ABB RobotStudio station: Paletizado.rspag

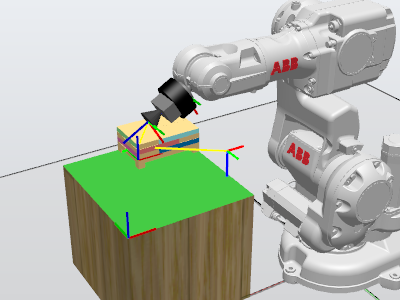
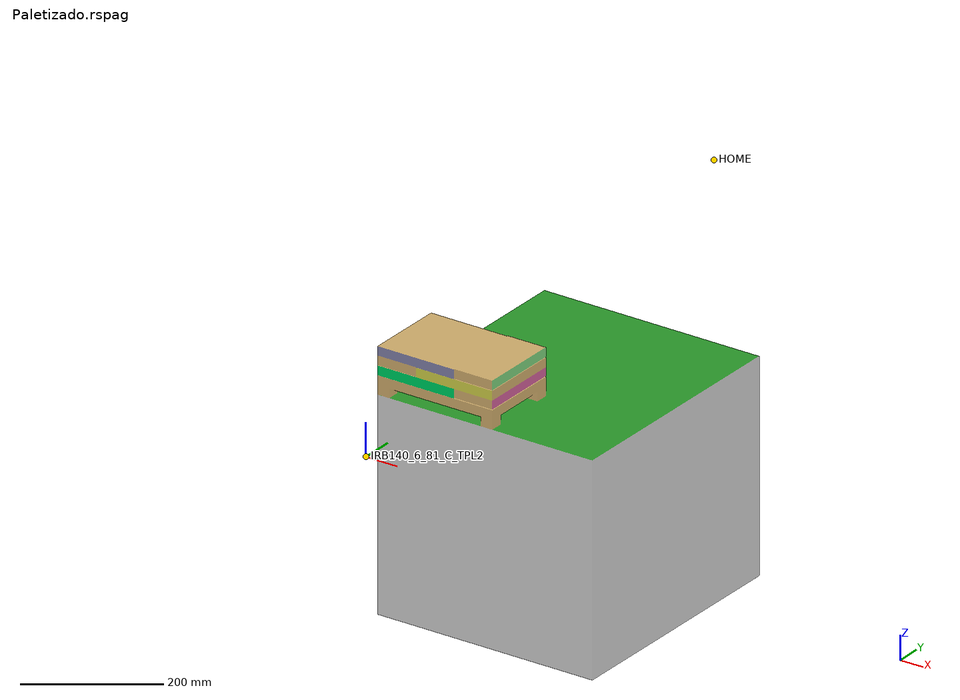
[picture v1: parts stored in the station drawn from their meshes, with robot base, taught points and paths (robot models come from the ABB library and are not in the file)]
--- station ---
Station Paletizado (saved by RobotStudio 25.1.11167.1)
Controller IRB140_6_81_TPL2
  mechanical unit ROB_1: IRB140_6_81_C_TPL2, 6 joints, base frame (0, 0, 0) mm
Layout (positions relative to the parent item):
  - Mesa [part], size 365 x 405 x 340 mm
  - Pallet [part], size 195 x 130 x 30 mm
  - Pieza1 [part] at (0, -275, 60) mm, size 130 x 65 x 15 mm
  - Pieza2 [part] at (729.91, -395, 45.09) mm, rotated rx 0 ry 0 rz 180 deg, size 130 x 65 x 15 mm
  - Pieza3 [part] at (490, 30, 30.97) mm, rotated rx 0 ry 0 rz -90 deg, size 130 x 65 x 15 mm
  - Pieza4 [part] at (795, -395, 0) mm, rotated rx 0 ry 0 rz -180 deg, size 130 x 65 x 15 mm
  - Pieza5 [part] at (65, -275, -15) mm, size 130 x 65 x 15 mm
  - Pieza6 [part] at (305, -700, -29.39) mm, rotated rx 0 ry 0 rz 90 deg, size 130 x 65 x 15 mm
  - Pieza7 [part] at (0, -275, -60) mm, size 130 x 65 x 15 mm
  - Pieza8 [part] at (729.88, -395, -74.88) mm, rotated rx 0 ry 0 rz 180 deg, size 130 x 65 x 15 mm
  - Pieza9 [part] at (490, 30, -88.74) mm, rotated rx 0 ry 0 rz -90 deg, size 130 x 65 x 15 mm
  - Sopapa [mechanism] at (506.29, 0, 679.5) mm, rotated rx 180 ry 60 rz 180 deg
      TCP Sopapa at (0, -5, 103) mm
      links: Sopapa
  - IRB140_6_81_C_TPL2 [mechanism, from %ABB.RobotStudio.Models.IRB140%\IRB140_6_81_C_G_03.rslib] at (0, 0, 0) mm; joint values [0, 0, 0, 0, 0.5236, 0] (rad or m)
Attachment: Sopapa is attached to IRB140_6_81_C_TPL2 / Link6
EventTableEntry 1212: Group=, Trigger=DO_Pinza 1213, Actions=[EventTableActionAttach 1214], Comment=, ActivationMode=2, Cyclic=false
EventTableTriggerIO 1213: IOValue=[1], IRC5Controller=? -1, Operator=0, SignalSource=? -1
EventTableActionAttach 1214: AttachmentParent=Sopapa 1252, AttachmentChild=? -1, MountObject=false, Offset=[X=1, Y=0, Z=0, W=0, X=0, Y=1, Z=0, W=0, X=0, Y=0, Z=1, W=0, X=0, Y=0, Z=0, W=1], FlangeIndext=0, FindNearest=true
EventTableEntry 1219: Group=, Trigger=DO_Pinza 1220, Actions=[EventTableActionDetach 1221], Comment=, ActivationMode=2, Cyclic=false
EventTableTriggerIO 1220: IOValue=[0], IRC5Controller=? -1, Operator=0, SignalSource=? -1
EventTableActionDetach 1221: AttachmentParent=Sopapa 1252, AttachmentChild=? -1
EventTableEntry 2390: Group=, Trigger=DO_SOPAPA 2391, Actions=[EventTableActionAttach 2392], Comment=, ActivationMode=2, Cyclic=false
EventTableTriggerIO 2391: IOValue=[1], IRC5Controller=? -1, Operator=0, SignalSource=IRB140_6_81_TPL2 1258
EventTableActionAttach 2392: AttachmentParent=Sopapa 1252, AttachmentChild=? -1, MountObject=false, Offset=[X=1, Y=0, Z=0, W=0, X=0, Y=1, Z=0, W=0, X=0, Y=0, Z=1, W=0, X=0, Y=0, Z=0, W=1], FlangeIndext=0, FindNearest=true
EventTableEntry 3475: Group=, Trigger=DO_SOPAPA 3476, Actions=[EventTableActionDetach 3477], Comment=, ActivationMode=2, Cyclic=false
EventTableTriggerIO 3476: IOValue=[0], IRC5Controller=? -1, Operator=0, SignalSource=IRB140_6_81_TPL2 1258
EventTableActionDetach 3477: AttachmentParent=Sopapa 1252, AttachmentChild=? -1
Targets, tools, work objects and paths stored in the station and not in the controller backup, written as RAPID:
! task T_ROB1
MODULE Module1
  CONST robtarget PPLACE1_2:=[[32.5,65,0],[0,0.707106781,0.707106781,0],[-1,0,-2,0],[9E+09,9E+09,9E+09,9E+09,9E+09,9E+09]];
  PROC Path_20()
    MoveL PPICK,v1000,z100,Sopapa\WObj:=RMESA;
    MoveL PPICK,v1000,z100,Sopapa\WObj:=RMESA;
    MoveL PPLACE1,v1000,z100,Sopapa\WObj:=RPALET;
    MoveL HOME,v1000,z100,Sopapa\WObj:=wobj0;
    MoveL PPLACE1_2,v1000,z100,Sopapa\WObj:=RPALET;
  ENDPROC
ENDMODULE


--- Backups/IRB140_6_81_TPL2/RAPID/TASK1/PROGMOD/CalibData.mod ---
MODULE CalibData
    TASK PERS wobjdata RPALET:=[FALSE,TRUE,"",[[495,-270,370],[0,0,0,1]],[[0,0,0],[1,0,0,0]]];
    TASK PERS wobjdata RMESA:=[FALSE,TRUE,"",[[665,5,340],[0,0,0,1]],[[0,0,0],[1,0,0,0]]];
ENDMODULE

--- Backups/IRB140_6_81_TPL2/RAPID/TASK1/PROGMOD/Module1.mod ---
MODULE Module1
    !!!!! USAR MAYUSCULAS PARA LAS CONSTANTES
    PERS tooldata Sopapa:=[TRUE,[[0,-5,103],[1,0,0,0]],[0.5,[0,0,40],[1,0,0,0],0,0,0]];
    PERS tooldata Sopapa_caja:=[TRUE,[[0,-5,118],[1,0,0,0]],[0.5,[0,0,40],[1,0,0,0],0,0,0]];
    CONST robtarget PPICK:=[[300,32.5,135],[0,1,0,0],[0,0,0,0],[9E+09,9E+09,9E+09,9E+09,9E+09,9E+09]];
    CONST robtarget PPLACE1:=[[32.5,65,0],[0,-0.707106781,0.707106781,0],[0,0,0,0],[9E+09,9E+09,9E+09,9E+09,9E+09,9E+09]];
    CONST robtarget HOME:=[[595.492267836,-5,628],[0.5,0,0.866025404,0],[0,-1,0,0],[9E+09,9E+09,9E+09,9E+09,9E+09,9E+09]];
    CONST num cant_cajas:=9;
    CONST num h_caja:=15;
    CONST num dx_PPLACE1:=130;
    VAR num CajasEnPalet:=0;

    !***********************************************************
    !
    ! Module:  Module1
    !
    ! Description:
    !   <Insert description here>
    !
    ! Author: CARLOS ISAAC
    !
    ! Version: 1.0
    !
    !***********************************************************


    !***********************************************************
    !
    ! Procedure main
    !
    !   This is the entry point of your program
    !
    !***********************************************************
    PROC main()
        !Add your code here
        VAR num pila:=0; !indica la pila actual de paletizado iniciando en 0
        VAR num caja_pilai:=0; !Contador de cajas en la pila i comienza en 0
        VAR num CajaEnPalet:=0;

        !FOR i FROM 0 TO cant_cajas-1 DO
        !   IF i MOD 3 = 0 AND i <> 0 THEN
        !        pila := pila +1; !cambio a la pilai
        !        caja_pilai:=0; !reinicio el contador de caja pues empiezo nueva pila
        !    ENDIF
        !    Pick(i*h_caja);
        !    Armar_pila(pila),(caja_pilai);
        !    caja_pilai:=caja_pilai + 1;
        !    CajasEnPalet := CajasEnPalet+1;
        !ENDFOR

        WHILE CajasEnPalet < cant_cajas DO
            IF CajasEnPalet MOD 3 = 0 AND CajasEnPalet <> 0 THEN
                pila := pila + 1;        ! Cambio a la pila siguiente
                caja_pilai := 0;         ! Reinicio el contador de cajas en la nueva pila
            ENDIF

            Pick(CajasEnPalet * h_caja);
            Armar_pila pila, caja_pilai;

            caja_pilai := caja_pilai + 1;
            CajasEnPalet := CajasEnPalet + 1;
        ENDWHILE

        !ENDWHILE

        MoveJ HOME,v100,fine,Sopapa\WObj:=wobj0;
    ENDPROC

    !Va variando la altura z donde busca la caja
    PROC Pick(num z)
        MoveJ Offs(PPICK, 0,0,30),v100,z10,Sopapa\WObj:=RMESA;
        MoveL Offs(PPICK,0,0,-z),v100,fine,Sopapa\WObj:=RMESA;
        SetDO DO_SOPAPA, 1;
        WaitTime(1);
        MoveL Offs(PPICK, 0, 0, 30),v100,z10,Sopapa\WObj:=RMESA;
    ENDPROC


    PROC Place(robtarget PPLACE, pos offset_PPLACE)
        MoveJ Offs(PPLACE, offset_PPLACE.x,offset_PPLACE.y,offset_PPLACE.z),v100,z10,Sopapa_caja\WObj:=RPALET;

        MoveL PPLACE,v50,fine,Sopapa_caja\WObj:=RPALET;
        SetDO DO_SOPAPA, 0;
        WaitTime(1);
        MoveL Offs(PPLACE,0,0,30),v100,z10,Sopapa\WObj:=RPALET;
    ENDPROC


    PROC Armar_pila(num pila, num caja_pilai)
        VAR num z;
        VAR robtarget PPLACE;
        VAR orient rotacion_place;
        !Desplazamientos respecto de PPLACE1 para pila tipo 1 (pila par)
        !VAR num d01{3} := [97.5,32.5,0]; !definirlo en funcion de dimensiones de la caja
        !VAR num d02{3} := [97.5,-32.5,0];
        VAR pos d01:=[97.5,32.5,0];
        VAR pos d02:=[97.5,-32.5,0];
        !Orientacion respecto RPALET para pila tipo 1 (pila par)
        VAR orient o1;
        VAR orient o2;
        !Offset de aproximación a PPLACE
        VAR pos offset_PPLACE := [0,0,30]; !El que es por defecto para PPLACE1
        !Para pila tipo 1 (par) offset para cada caja 1 y 2
        !VAR num offset_PPLACE_1{3} := [30,0,30];
        !VAR num offset_PPLACE_2{3} := [30,-30,30];
        VAR pos offset_PPLACE_1:=[30,0,30];
        VAR pos offset_PPLACE_2:=[30,-30,30];


        z := pila*h_caja;
        PPLACE:=Offs(PPLACE1,0,0,pila*h_caja); !Inicio la variable place y le doy la altura de la pila
        rotacion_place:=OrientZYX(90,0,180);
        o1:= OrientZYX(0,180,0);
        o2:= OrientZYX(0,0,180);

        IF pila MOD 2 <> 0 THEN !pila impar modifico a a otra forma
            PPLACE:=Offs(PPLACE,dx_PPLACE1,0,0);
            PPLACE.rot:=rotacion_place; !creo que esta tmb es correcta y queda mejor calcularla así
            !PPLACE.rot:=[0,0.707106781,0.707106781,0]; !Orientación correcta verificada
            d01 := [-97.5,-32.5,0];
            d02 := [-97.5,32.5,0];
            o1:=OrientZYX(0,0,180);
            o2:=OrientZYX(0,180,0);
            offset_PPLACE_1 := [-30,0,30];
            offset_PPLACE_2 := [-30,30,30];
        ENDIF

        IF caja_pilai = 1 THEN
            PPLACE:=Offs(PPLACE,d01.x,d01.y,d01.z);
            PPLACE.rot:=o1;
            offset_PPLACE := offset_PPLACE_1;
        ELSEIF caja_pilai = 2 THEN
            PPLACE:=Offs(PPLACE,d02.x,d02.y,d02.z);
            PPLACE.rot:=o2;
            offset_PPLACE := offset_PPLACE_2;
        ENDIF

        Place(PPLACE),(offset_PPLACE);
    ENDPROC
ENDMODULE

--- Backups/IRB140_6_81_TPL2/SYSPAR/EIO.cfg ---
EIO:CFG_1.0:6:1::
#
EIO_SIGNAL:

      -Name "DO_SOPAPA" -SignalType "DO" -Label "0" -Access "All"
